% RSLogix 500 project LAB 10 done.RSS, saved by version 8.30.00.16 %
PROJECT "UNTITLED"    % processor: MicroLogix 1000 %

PROGRAM FILES
  LAD 2 "MAIN_PROG"  17 rungs
  LAD 3 "USER_FAULT"  1 rungs
  LAD 4 "HSC_INT"  1 rungs
  LAD 5 "STI_INT"  1 rungs
  LAD 6, 7, 8, 9, 10, 11, 12, 13, 14, 15, 16: only END

DATA FILES
  O0 OUTPUT  1 elements
  I1 INPUT  2 elements
  S2 STATUS  33 elements
  B3 BINARY  32 elements
  T4 TIMER  40 elements
  C5 COUNTER  32 elements
  R6 CONTROL  16 elements
  N7 INTEGER  105 elements

LADDER 2 "MAIN_PROG"
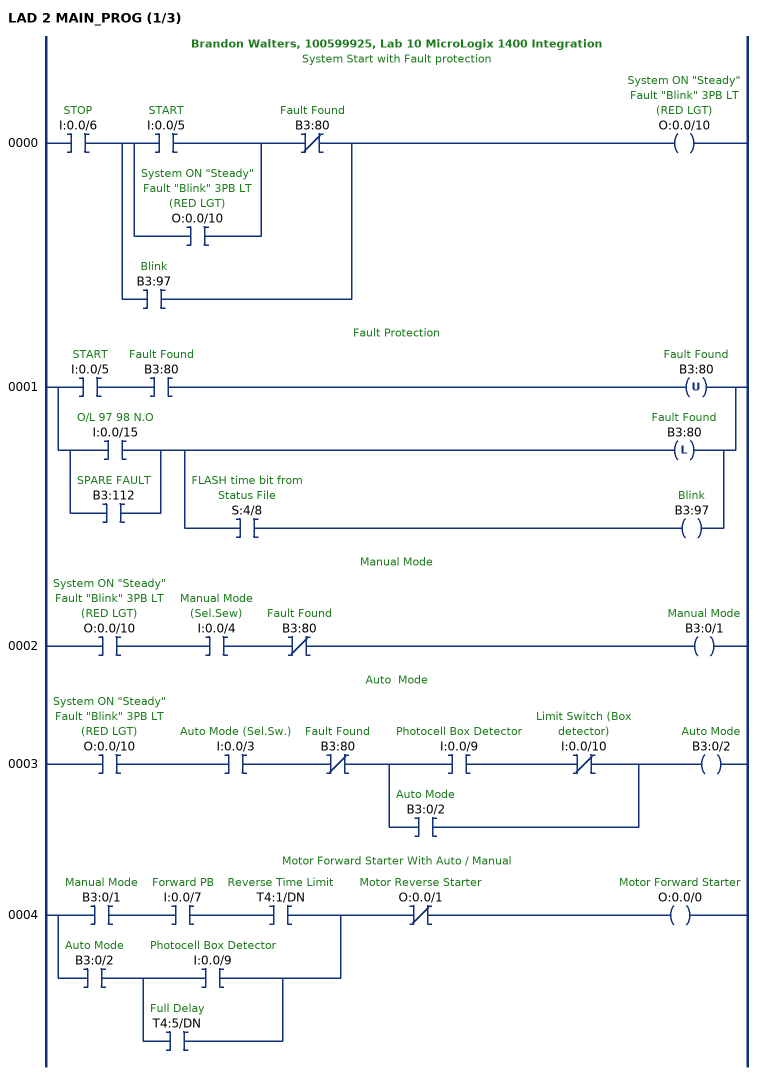
% Rung: 0 %  % edit flag set %
% TITLE: Brandon Walters, 100599925, Lab 10 MicroLogix 1400 Integration %
% System Start with Fault protection %
SOR XIC I:0.0/6 BST BST XIC I:0.0/5 NXB XIC O:0.0/10 BND XIO B3:80 NXB XIC B3:97 BND OTE O:0.0/10 EOR
%   I:0.0/6  "STOP" %
%   I:0.0/5  "START" %
%   O:0.0/10  "System ON "Steady" Fault "Blink" 3PB LT (RED LGT)" %
%   B3:80  "Fault Found" %
%   B3:97  "Blink" %
% Rung: 1 %  % edit flag set %
% Fault Protection %
SOR BST XIC I:0.0/5 XIC B3:80 OTU B3:80 NXB BST XIC I:0.0/15 NXB XIC B3:112 BND BST OTL B3:80 NXB XIC S:4/8 OTE B3:97 BND BND EOR
%   I:0.0/5  "START" %
%   B3:80  "Fault Found" %
%   I:0.0/15  "O/L 97 98 N.O" %
%   B3:112  "SPARE FAULT" %
%   S:4/8  "FLASH time bit from Status File" %
%   B3:97  "Blink" %
% Rung: 2 %  % edit flag set %
% Manual Mode %
SOR XIC O:0.0/10 XIC I:0.0/4 XIO B3:80 OTE B3:0/1 EOR
%   O:0.0/10  "System ON "Steady" Fault "Blink" 3PB LT (RED LGT)" %
%   I:0.0/4  "Manual Mode (Sel.Sew)" %
%   B3:80  "Fault Found" %
%   B3:0/1  "Manual Mode" %
% Rung: 3 %  % edit flag set %
% Auto  Mode %
SOR XIC O:0.0/10 XIC I:0.0/3 XIO B3:80 BST XIC I:0.0/9 XIO I:0.0/10 NXB XIC B3:0/2 BND OTE B3:0/2 EOR
%   O:0.0/10  "System ON "Steady" Fault "Blink" 3PB LT (RED LGT)" %
%   I:0.0/3  "Auto Mode (Sel.Sw.)" %
%   B3:80  "Fault Found" %
%   I:0.0/9  "Photocell Box Detector" %
%   I:0.0/10  "Limit Switch (Box detector)" %
%   B3:0/2  "Auto Mode" %
% Rung: 4 %  % edit flag set %
% Motor Forward Starter With Auto / Manual %
SOR BST XIC B3:0/1 XIC I:0.0/7 XIC T4:1/DN NXB XIC B3:0/2 BST XIC I:0.0/9 NXB XIC T4:5/DN BND BND XIO O:0.0/1 OTE O:0.0/0 EOR
%   B3:0/1  "Manual Mode" %
%   I:0.0/7  "Forward PB" %
%   T4:1  "Reverse Time Limit" %
%   B3:0/2  "Auto Mode" %
%   I:0.0/9  "Photocell Box Detector" %
%   T4:5  "Full Delay" %
%   O:0.0/1  "Motor Reverse Starter" %
%   O:0.0/0  "Motor Forward Starter" %

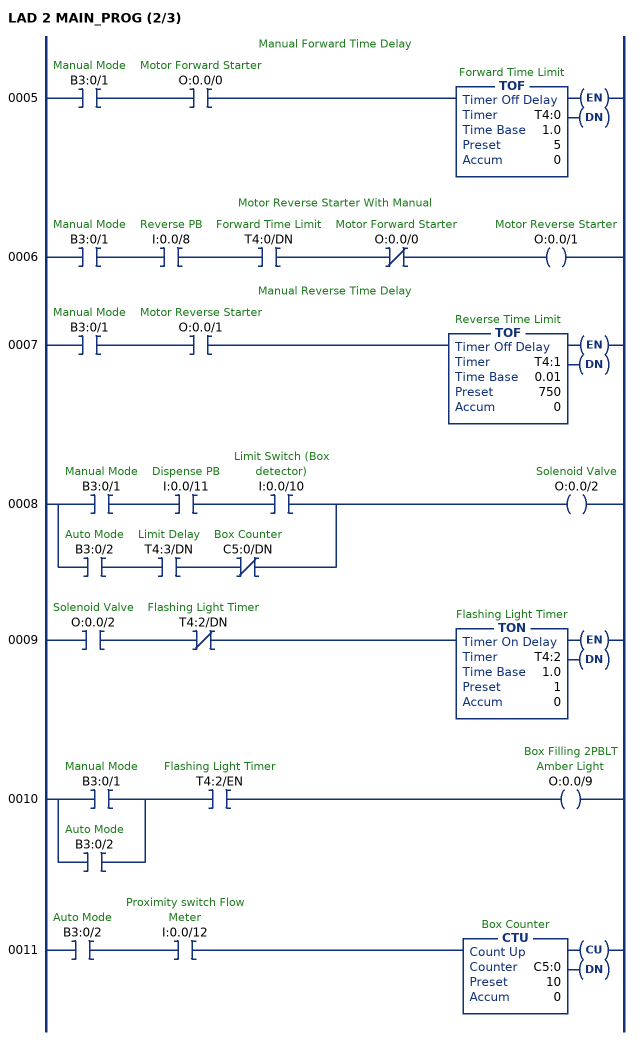
% Rung: 5 %  % edit flag set %
% Manual Forward Time Delay %
SOR XIC B3:0/1 XIC O:0.0/0 TOF T4:0 1.0 5 0 EOR
%   B3:0/1  "Manual Mode" %
%   O:0.0/0  "Motor Forward Starter" %
%   T4:0  "Forward Time Limit" %
% Rung: 6 %  % edit flag set %
% Motor Reverse Starter With Manual %
SOR XIC B3:0/1 XIC I:0.0/8 XIC T4:0/DN XIO O:0.0/0 OTE O:0.0/1 EOR
%   B3:0/1  "Manual Mode" %
%   I:0.0/8  "Reverse PB" %
%   T4:0  "Forward Time Limit" %
%   O:0.0/0  "Motor Forward Starter" %
%   O:0.0/1  "Motor Reverse Starter" %
% Rung: 7 %  % edit flag set %
% Manual Reverse Time Delay %
SOR XIC B3:0/1 XIC O:0.0/1 TOF T4:1 0.01 750 0 EOR
%   B3:0/1  "Manual Mode" %
%   O:0.0/1  "Motor Reverse Starter" %
%   T4:1  "Reverse Time Limit" %
% Rung: 8 %  % edit flag set %
SOR BST XIC B3:0/1 XIC I:0.0/11 XIC I:0.0/10 NXB XIC B3:0/2 XIC T4:3/DN XIO C5:0/DN BND OTE O:0.0/2 EOR
%   B3:0/1  "Manual Mode" %
%   I:0.0/11  "Dispense PB" %
%   I:0.0/10  "Limit Switch (Box detector)" %
%   B3:0/2  "Auto Mode" %
%   T4:3  "Limit Delay" %
%   C5:0  "Box Counter" %
%   O:0.0/2  "Solenoid Valve" %
% Rung: 9 %  % edit flag set %
SOR XIC O:0.0/2 XIO T4:2/DN TON T4:2 1.0 1 0 EOR
%   O:0.0/2  "Solenoid Valve" %
%   T4:2/DN  "Flashing Light Timer" %
%   T4:2  "Flashing Light Timer" %
% Rung: 10 %  % edit flag set %
SOR BST XIC B3:0/1 NXB XIC B3:0/2 BND XIC T4:2/EN OTE O:0.0/9 EOR
%   B3:0/1  "Manual Mode" %
%   B3:0/2  "Auto Mode" %
%   T4:2/EN  "Flashing Light Timer" %
%   O:0.0/9  "Box Filling 2PBLT Amber Light" %
% Rung: 11 %  % edit flag set %
SOR XIC B3:0/2 XIC I:0.0/12 CTU C5:0 10 0 EOR
%   B3:0/2  "Auto Mode" %
%   I:0.0/12  "Proximity switch Flow Meter" %
%   C5:0  "Box Counter" %

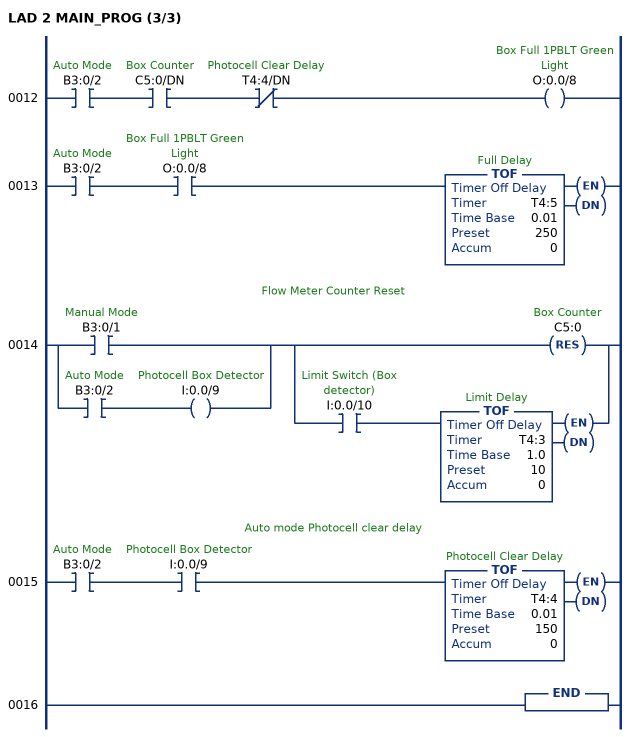
% Rung: 12 %  % edit flag set %
SOR XIC B3:0/2 XIC C5:0/DN XIO T4:4/DN OTE O:0.0/8 EOR
%   B3:0/2  "Auto Mode" %
%   C5:0  "Box Counter" %
%   T4:4  "Photocell Clear Delay" %
%   O:0.0/8  "Box Full 1PBLT Green Light" %
% Rung: 13 %  % edit flag set %
SOR XIC B3:0/2 XIC O:0.0/8 TOF T4:5 0.01 250 0 EOR
%   B3:0/2  "Auto Mode" %
%   O:0.0/8  "Box Full 1PBLT Green Light" %
%   T4:5  "Full Delay" %
% Rung: 14 %  % edit flag set %
% Flow Meter Counter Reset %
SOR BST XIC B3:0/1 NXB XIC B3:0/2 OTE I:0.0/9 BND BST RES C5:0 NXB XIC I:0.0/10 TOF T4:3 1.0 10 0 BND EOR
%   B3:0/1  "Manual Mode" %
%   B3:0/2  "Auto Mode" %
%   I:0.0/9  "Photocell Box Detector" %
%   OTE I:0.0/9  "One Shot" %
%   C5:0  "Box Counter" %
%   I:0.0/10  "Limit Switch (Box detector)" %
%   T4:3  "Limit Delay" %
% Rung: 15 %  % edit flag set %
% Auto mode Photocell clear delay %
SOR XIC B3:0/2 XIC I:0.0/9 TOF T4:4 0.01 150 0 EOR
%   B3:0/2  "Auto Mode" %
%   I:0.0/9  "Photocell Box Detector" %
%   T4:4  "Photocell Clear Delay" %
% Rung: 16 %
SOR END EOR
